FUNCTION_BLOCK TestUtils EXTENDS TcUnit.FB_TestSuite
VAR_INPUT
END_VAR
VAR_OUTPUT
END_VAR
VAR
END_VAR

test_remove_project_from_path();

METHOD test_remove_project_from_path
VAR
  path: STRING(255);
END_VAR
TEST('Test remove project from path');

path := 'project.project.MAIN.test';

AssertEquals_STRING('MAIN.test', remove_project_from_path(path), '');

TEST_FINISHED();
END_METHOD

END_FUNCTION_BLOCK

(* stored: Version 1.1.0.1, ProductVersion 3.1.4024.9
   POU TestUtils: Id {3fa20875-225a-4206-a46a-7351023bbda0}, SpecialFunc None
   Method test_remove_project_from_path: Id {e8007b6e-7292-4cc4-be66-05706e700c47} *)
